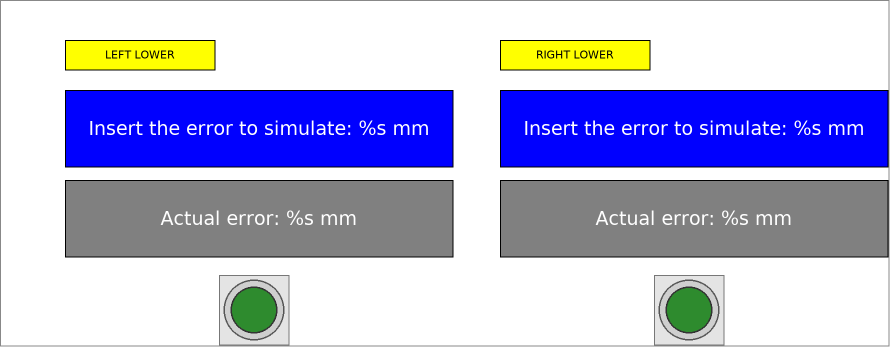
VISUALIZATION CARTON_FEEDING_TOOTH_DISTANCE  // 890x347
    Rectangle (65,40 150x30), "LEFT LOWER"
    Rectangle (500,40 150x30), "RIGHT LOWER"
    RoundedRectangle (65,90 388x77), "Insert the error to simulate: %s mm", text variable: wu_cartonFeeding_leftSide_toothDistance.simulation_error
        OnMouseUp: write the text variable via VisuDialogs.Numpad
    RoundedRectangle (500,90 388x77), "Insert the error to simulate: %s mm", text variable: wu_cartonFeeding_rightSide_toothDistance.simulation_error
        OnMouseUp: write the text variable via VisuDialogs.Numpad
    RoundedRectangle (65,180 388x77), "Actual error: %s mm", text variable: wu_cartonFeeding_leftSide_toothDistance.simulation_error_current_value_visu
        OnMouseUp: write the text variable via VisuDialogs.Numpad
    RoundedRectangle (500,180 388x77), "Actual error: %s mm", text variable: wu_cartonFeeding_rightSide_toothDistance.simulation_error_current_value_visu
        OnMouseUp: write the text variable via VisuDialogs.Numpad
    PushSwitch (219,275 70x70), variable: wu_cartonFeeding_leftSide_toothDistance.simulation_error_download, behaviour: TAP, style: Switch-PushSwitch-Green
    PushSwitch (654,275 70x70), variable: wu_cartonFeeding_rightSide_toothDistance.simulation_error_download, behaviour: TAP, style: Switch-PushSwitch-Green
END_VISUALIZATION

(* stored: Version 1.1.0.1, ProductVersion 3.1.4024.3
   Visu CARTON_FEEDING_TOOTH_DISTANCE: Id {6d8ab176-8153-451d-aec3-12c6946cfa90} *)
